TYPE ST_state_machine_com :
STRUCT
	Car_state_machine:INT;
	Arm1_state_machine:INT;
	Arm2_state_machine:INT;
	Arm3_state_machine:INT;
	Arm4_state_machine:INT;
END_STRUCT
END_TYPE

(* stored: Version 1.1.0.1, ProductVersion 3.1.4024.11
   DUT ST_state_machine_com: Id {eacf3ae3-4e42-4e69-9949-1ccf58239b23} *)
